// TIA Portal V19 export
FUNCTION "FC_Reset_FWBits_im_Bad" : Void   // FC18, STL
{ S7_Optimized_Access := 'FALSE' }
AUTHOR : MS
// Setzt die Bits "FW über Bad" und "FW kommt"zurück
// stored: AutoNumber false
   VAR_INPUT
      Reset_in_out_nen : Bool;
   END_VAR
   VAR_TEMP
      anzahl : Int;
      count : Int;
      first : Bool;
   END_VAR
BEGIN

NETWORK
TITLE = 
// Schleife über alle Badpositionen
      L     "DB_ANLAGE".config.ANZ_Pos;
ret:  T     #anzahl;
      L     "DB_POS".LENG;
      *I;
      L     "DB_POS".Offset;
      +I;
      SLD   3;
      LAR1;
      OPN   "DB_POS";
//vor Bearbeitung FWs
      AN    #Reset_in_out_nen;
      R     DBX [AR1, P#6.4];  //FW kommt
      R     DBX [AR1, P#6.5];  //FW in Pos
      R     DBX [AR1, P#6.6];  //FW hebt
      R     DBX [AR1, P#6.7];  //FW senkt
//nach Bearbeitung FWs
      AN    #Reset_in_out_nen;
      JC    noGR;
      OPN   "DB_POS";
      R     DBX [AR1, P#7.3];  //FW Badbedienung nicht möglich
      R     DBX [AR1, P#96.6];  //"DB_POS".POS[0].Expo_Off
      S     #first;

noGR: L     #anzahl;
      L     1;
      <=I;
      BEC;
      L     #anzahl;
      L     1;
      -I;
      JU    ret;

END_FUNCTION
